// TIA Portal V20 export
TYPE "typeSequenceControlNode_sideTapeLoading"
// stored: Namespace Unit1.Em4
   STRUCT
      jobs : "LAF_typeJobs";
      sequence : "LAF_typeSequence";
      selectJobStatus { S7_SetPoint := 'True'} : Array[0..10] of "LAF_typeJobStatus";
      "step" : "LER_typeStep";
      jobInterface : "Unit1.Em4.typeSequenceControlNodeJobInterface_sideTapeLoading";
      homeCheck : "Unit1.Em4.typeSequenceControlNodeHomeCheck_sideTapeLoading";
   END_STRUCT;
   // // "step".action1[101] : Step[101] : JOB[1] Condition
   // // "step".action1[110] : Step[110] : Side Tape Loading Down
   // // "step".action1[120] : Step[120] : Side Tape Clamp Open
   // // "step".action1[130] : Step[130] : Side Tape Cutter Backward
   // // "step".action1[140] : Step[140] : Side Tape Cutter Clamp Forward
   // // "step".action1[150] : Step[150] : Side Tape Tension Backward
   // // "step".action1[190] : Step[190] : JOB[1] Step End
   // // "step".action1[201] : Step[201] : JOB[2] Condition
   // // "step".action1[210] : Step[210] : Side Tape Loading Up, Tension Backward
   // // "step".action1[220] : Step[220] : Side Tape Clamp Close
   // // "step".action1[230] : Step[230] : Side Tape Cutter Clamp Backward
   // // "step".action1[240] : Step[240] : Side Tape Loading Down, Tension Forward
   // // "step".action1[250] : Step[250] : Side Tape Cutter Clamp Forward
   // // "step".action1[260] : Step[260] : Side Tape Tension Backward
   // // "step".action1[290] : Step[290] : JOB[2] Step End
   // // "step".transition1[101] : Step[101] : JOB[1] Condition
   // // "step".transition1[110] : Step[110] : Side Tape Loading Down
   // // "step".transition1[120] : Step[120] : Side Tape Clamp Open
   // // "step".transition1[130] : Step[130] : Side Tape Cutter Backward
   // // "step".transition1[140] : Step[140] : Side Tape Cutter Clamp Forward
   // // "step".transition1[150] : Step[150] : Side Tape Tension Backward
   // // "step".transition1[190] : Step[190] : JOB[1] Step End
   // // "step".transition1[201] : Step[201] : JOB[2] Condition
   // // "step".transition1[210] : Step[210] : Side Tape Loading Up, Tension Backward
   // // "step".transition1[220] : Step[220] : Side Tape Clamp Close
   // // "step".transition1[230] : Step[230] : Side Tape Cutter Clamp Backward
   // // "step".transition1[240] : Step[240] : Side Tape Loading Down, Tension Forward
   // // "step".transition1[250] : Step[250] : Side Tape Cutter Clamp Forward
   // // "step".transition1[260] : Step[260] : Side Tape Tension Backward
   // // "step".transition1[290] : Step[290] : JOB[2] Step End
END_TYPE
